# EPICS substitutions: ek9000App/Db/EL1034.substitutions
file EL1034.template
{ 	pattern
	{
		TERMINAL,

	}
	{
	}
}
